(* Schneider Machine Expert - Basic project PRAUT, file version 2.7.0.0 *)
(* ProjectInformations: Name=Nuevo proyecto *)

HARDWARE
  Cpu 0: TM221M16R/G
  EthernetConfiguration: NetworkName=M221, IpAllocationMode=FixedAddress, IpAddress=0.0.0.0, SubnetMask=0.0.0.0
  SerialLineConfiguration: Baud=Baud19200, Parity=ParityEven, DataBits=DataBits8, StopBits=StopBits1, PhysicalMedium=PhysicalMediumRs485, TransmissionMode=TransmissionModeModbusRtu, SlaveId=1, Addressing=SlaveAddressing
  MastTask: UsePeriodScanMode=false, PeriodScan=100
  FastTask: Period=255
  CpuBehavior: StartingMode=StartAsPreviousState, AutoSaveRamOnEeprom=true, WatchdogPeriod=250

SYMBOLS  (address, symbol, comment, settings)
  %M0       INICIO
  %M1       RESET
  %M2       STOP
  %M6       SCADA_GAB
  %M7       STOP_SCADA
  %M8       START_SCADA
  %M9       RESET_SCADA
  %M10      RESET_IO
  %M11      PILOTO
  %M20      START_LIGHT
  %M21      RESET_LIGHT
  %M22      STOP_LIGHT
  %M23      FACTORY_RESET
  %M40      OPERACION
  %MD0      LEVEL_METER
  %MD4      SETPOINT
  %MD6      SP_DISCHARGE
  %MD20     FILL_VALVE
  %MD22     DISCHARGE_VALVE
  %MD24     SP
  %MD26     PV
  %MD28     DV
  %MD29     NIVEL_TAN2
  %MD40     ERROR_LEVEL
  %MD42     ACUMULADOR
  %MD44     TOTAL_INTEGRAL
  %MD46     INTEGRAL
  %MD48     SET_LEVEL_SCADA
  %MD50     SET_DISCHARGE_SCADA
  %MD52     PI
  %TM0      T_INTEGRAL  [Preset=5, Base=OneSecond]

POU Nuevo POU
  (* SectionNumber=1 *)

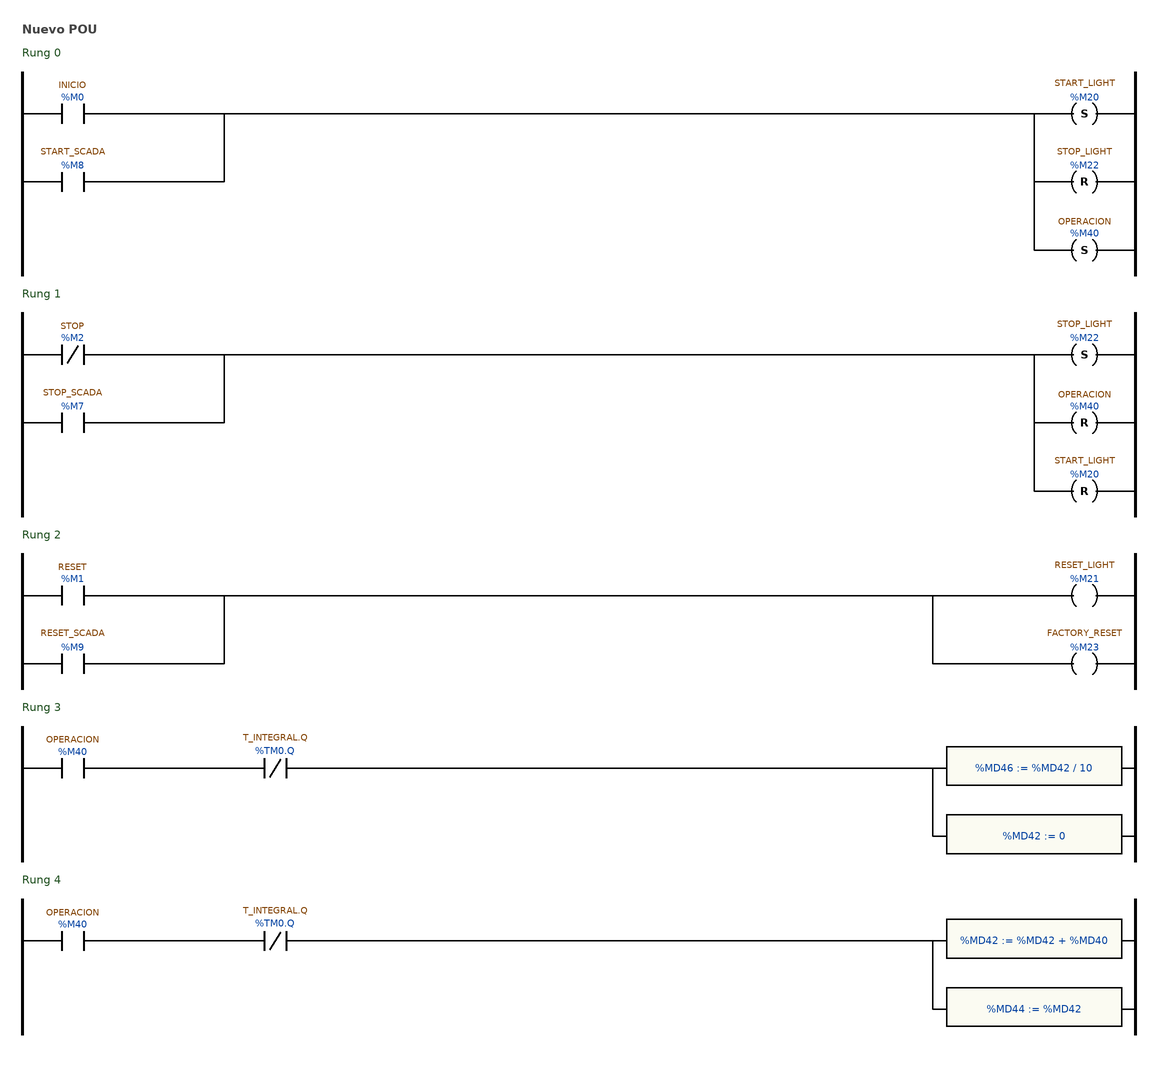

// Rung 0
  LD %M0                  (* INICIO *)
  OR %M8                  (* START_SCADA *)
  S %M20                  (* START_LIGHT *)
  R %M22                  (* STOP_LIGHT *)
  S %M40                  (* OPERACION *)
  // as ST:
  //   IF INICIO OR START_SCADA THEN START_LIGHT := TRUE; END_IF;
  //   IF INICIO OR START_SCADA THEN STOP_LIGHT := FALSE; END_IF;
  //   IF INICIO OR START_SCADA THEN OPERACION := TRUE; END_IF;

// Rung 1
  LDN %M2                 (* STOP *)
  OR %M7                  (* STOP_SCADA *)
  S %M22                  (* STOP_LIGHT *)
  R %M40                  (* OPERACION *)
  R %M20                  (* START_LIGHT *)
  // as ST:
  //   IF NOT STOP OR STOP_SCADA THEN STOP_LIGHT := TRUE; END_IF;
  //   IF NOT STOP OR STOP_SCADA THEN OPERACION := FALSE; END_IF;
  //   IF NOT STOP OR STOP_SCADA THEN START_LIGHT := FALSE; END_IF;

// Rung 2
  LD %M1                  (* RESET *)
  OR %M9                  (* RESET_SCADA *)
  ST %M21                 (* RESET_LIGHT *)
  ST %M23                 (* FACTORY_RESET *)
  // as ST:
  //   RESET_LIGHT := RESET OR RESET_SCADA;
  //   FACTORY_RESET := RESET OR RESET_SCADA;

// Rung 3
  LD %M40                 (* OPERACION *)
  ANDN %TM0.Q             (* T_INTEGRAL *)
  [ %MD46 := %MD42 / 10 ] (* INTEGRAL, ACUMULADOR *)
  [ %MD42 := 0 ]          (* ACUMULADOR *)
  // as ST:
  //   IF OPERACION AND NOT T_INTEGRAL.Q THEN INTEGRAL := ACUMULADOR / 10; END_IF;
  //   IF OPERACION AND NOT T_INTEGRAL.Q THEN ACUMULADOR := 0; END_IF;

// Rung 4
  LD %M40                 (* OPERACION *)
  ANDN %TM0.Q             (* T_INTEGRAL *)
  [ %MD42 := %MD42 + %MD40 ](* ACUMULADOR, ACUMULADOR, ERROR_LEVEL *)
  [ %MD44 := %MD42 ]      (* TOTAL_INTEGRAL, ACUMULADOR *)
  // as ST:
  //   IF OPERACION AND NOT T_INTEGRAL.Q THEN ACUMULADOR := ACUMULADOR + ERROR_LEVEL; END_IF;
  //   IF OPERACION AND NOT T_INTEGRAL.Q THEN TOTAL_INTEGRAL := ACUMULADOR; END_IF;

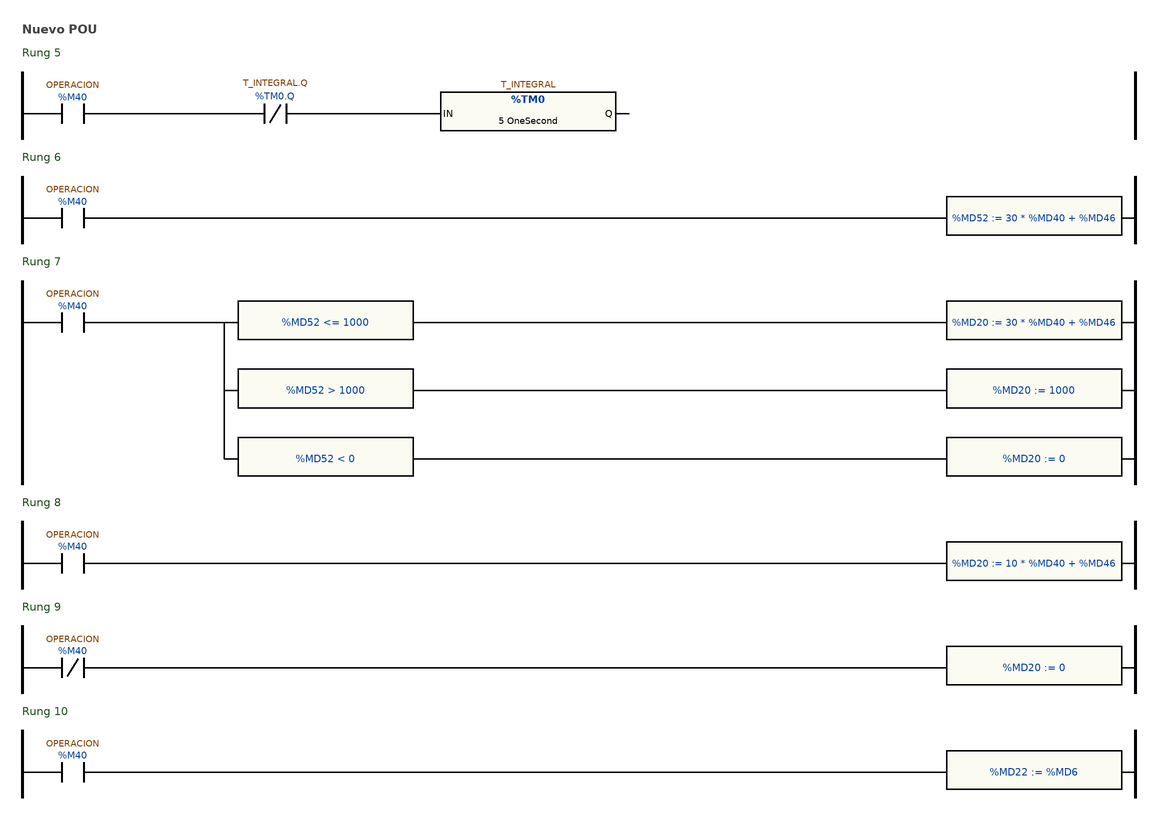

// Rung 5
  BLK %TM0                (* T_INTEGRAL *)
  LD %M40                 (* OPERACION *)
  ANDN %TM0.Q             (* T_INTEGRAL *)
  IN
  END_BLK
  // as ST:
  //   T_INTEGRAL(IN := OPERACION AND NOT T_INTEGRAL.Q);

// Rung 6
  LD %M40                 (* OPERACION *)
  [ %MD52 := 30 * %MD40 + %MD46 ](* PI, ERROR_LEVEL, INTEGRAL *)
  // as ST:
  //   IF OPERACION THEN PI := 30 * ERROR_LEVEL + INTEGRAL; END_IF;

// Rung 7
  LD %M40                 (* OPERACION *)
  MPS
  AND [ %MD52 <= 1000 ]   (* PI *)
  [ %MD20 := 30 * %MD40 + %MD46 ](* FILL_VALVE, ERROR_LEVEL, INTEGRAL *)
  MRD
  AND [ %MD52 > 1000 ]    (* PI *)
  [ %MD20 := 1000 ]       (* FILL_VALVE *)
  MPP
  AND [ %MD52 < 0 ]       (* PI *)
  [ %MD20 := 0 ]          (* FILL_VALVE *)
  // as ST:
  //   IF OPERACION AND PI <= 1000 THEN FILL_VALVE := 30 * ERROR_LEVEL + INTEGRAL; END_IF;
  //   IF OPERACION AND PI > 1000 THEN FILL_VALVE := 1000; END_IF;
  //   IF OPERACION AND PI < 0 THEN FILL_VALVE := 0; END_IF;

// Rung 8
  LD %M40                 (* OPERACION *)
  [ %MD20 := 10 * %MD40 + %MD46 ](* FILL_VALVE, ERROR_LEVEL, INTEGRAL *)
  // as ST:
  //   IF OPERACION THEN FILL_VALVE := 10 * ERROR_LEVEL + INTEGRAL; END_IF;

// Rung 9
  LDN %M40                (* OPERACION *)
  [ %MD20 := 0 ]          (* FILL_VALVE *)
  // as ST:
  //   IF NOT OPERACION THEN FILL_VALVE := 0; END_IF;

// Rung 10
  LD %M40                 (* OPERACION *)
  [ %MD22 := %MD6 ]       (* DISCHARGE_VALVE, SP_DISCHARGE *)
  // as ST:
  //   IF OPERACION THEN DISCHARGE_VALVE := SP_DISCHARGE; END_IF;

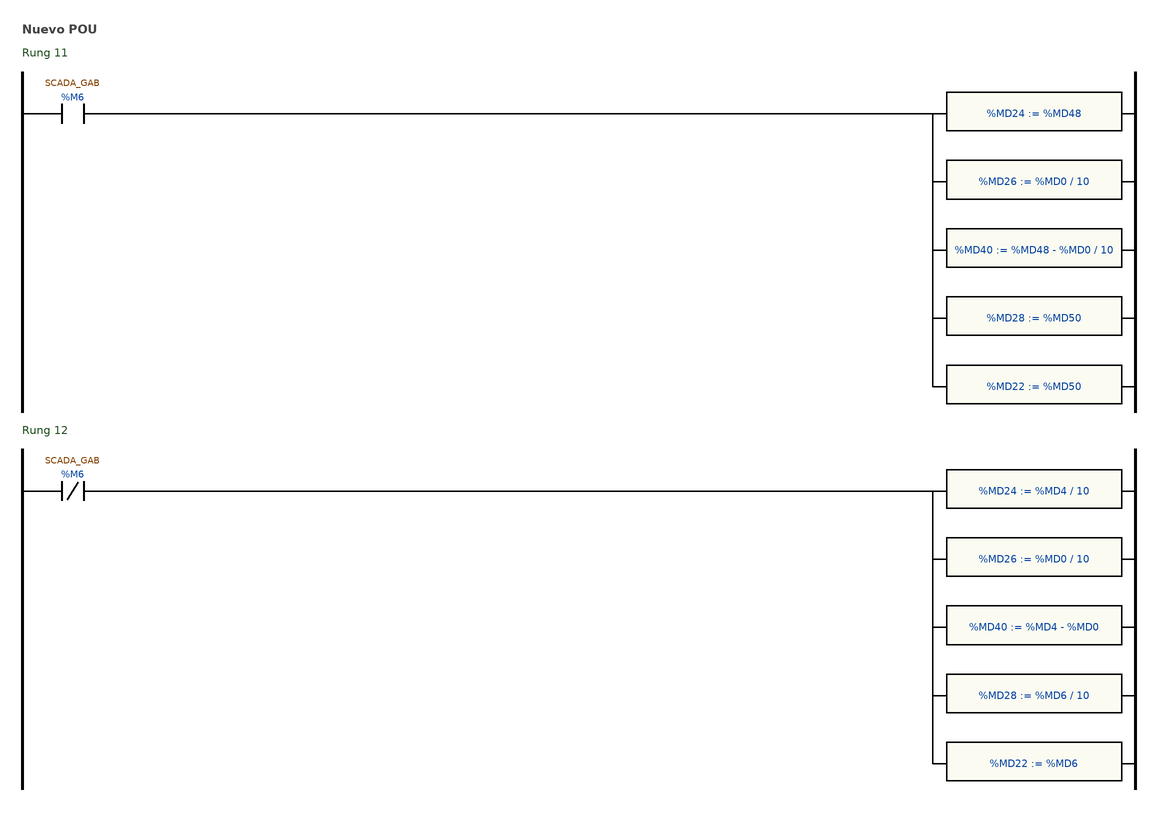

// Rung 11
  LD %M6                  (* SCADA_GAB *)
  [ %MD24 := %MD48 ]      (* SP, SET_LEVEL_SCADA *)
  [ %MD26 := %MD0 / 10 ]  (* PV, LEVEL_METER *)
  [%MD40 := %MD48 - %MD0 / 10](* ERROR_LEVEL, SET_LEVEL_SCADA, LEVEL_METER *)
  [ %MD28 := %MD50 ]      (* DV, SET_DISCHARGE_SCADA *)
  [ %MD22 := %MD50 ]      (* DISCHARGE_VALVE, SET_DISCHARGE_SCADA *)
  // as ST:
  //   IF SCADA_GAB THEN SP := SET_LEVEL_SCADA; END_IF;
  //   IF SCADA_GAB THEN PV := LEVEL_METER / 10; END_IF;
  //   IF SCADA_GAB THEN ERROR_LEVEL := SET_LEVEL_SCADA - LEVEL_METER / 10; END_IF;
  //   IF SCADA_GAB THEN DV := SET_DISCHARGE_SCADA; END_IF;
  //   IF SCADA_GAB THEN DISCHARGE_VALVE := SET_DISCHARGE_SCADA; END_IF;

// Rung 12
  LDN %M6                 (* SCADA_GAB *)
  [ %MD24 := %MD4 / 10 ]  (* SP, SETPOINT *)
  [ %MD26 := %MD0 / 10 ]  (* PV, LEVEL_METER *)
  [ %MD40 := %MD4 - %MD0 ](* ERROR_LEVEL, SETPOINT, LEVEL_METER *)
  [ %MD28 := %MD6 / 10 ]  (* DV, SP_DISCHARGE *)
  [ %MD22 := %MD6 ]       (* DISCHARGE_VALVE, SP_DISCHARGE *)
  // as ST:
  //   IF NOT SCADA_GAB THEN SP := SETPOINT / 10; END_IF;
  //   IF NOT SCADA_GAB THEN PV := LEVEL_METER / 10; END_IF;
  //   IF NOT SCADA_GAB THEN ERROR_LEVEL := SETPOINT - LEVEL_METER; END_IF;
  //   IF NOT SCADA_GAB THEN DV := SP_DISCHARGE / 10; END_IF;
  //   IF NOT SCADA_GAB THEN DISCHARGE_VALVE := SP_DISCHARGE; END_IF;
